{attribute 'GeneratedUsingTerminal: EJ9001-0000-0016'}
{attribute addProperty BoxType "EJ9001-0000-0016"}
{attribute addProperty Id "InfoDataAT %I*InfoData_6F19DB2B2"}
{attribute addProperty CRC "532711307"}
{attribute addProperty Size "2"}
TYPE EJ9001_1FC0878B :
STRUCT
	{attribute addProperty Name "InfoData"}
	InfoData : InfoData_6F19DB2B;
END_STRUCT
END_TYPE

(* stored: Version 1.2.0.0, ProductVersion 3.1.4024.9
   DUT EJ9001_1FC0878B: Id {c244f710-600a-41b6-9079-215443cd9097} *)
